PROGRAM PersonnelDoor
VAR
	
END_VAR

IF GVL_Doors.QQ1.OpenButtonRequestInput THEN
	GVL_Doors.QQ1.AccessAreaRequest := 1;
	GVL_Doors.QQ1.OpenButtonLED_Output := 1;
	GVL_Doors.QQ1.OkToUnlockDoor := 1; //Remove this once ventalation is hooked up. Ventalation and styrene sensor level will determine when this gets turned on.
	ELSE
	GVL_Doors.QQ1.OpenButtonLED_Output := 0;
END_IF

GVL_Doors.QQ1.OkToUnlockDoorRTRIG(CLK := GVL_Doors.QQ1.OkToUnlockDoor);


IF GVL_Doors.QQ1.OkToUnlockDoorRTRIG.Q THEN
	GVL_Doors.QQ1.AccessAreaRequest := 0;
	GVL_Doors.QQ1.OpenButtonLED_Output := 0;
	GVL_Doors.QQ1.LockButtonLED_Output := 1;
	GVL_Doors.QQ1.LockOutput := 1;
END_IF

IF GVL_Doors.QQ1.LockButtonRequestInput THEN
	GVL_Doors.QQ1.LockOutput := 0;	
	GVL_Doors.QQ1.LockButtonLED_Output := 0;
	GVL_Doors.QQ1.OkToUnlockDoor := 0; //Remove this once ventalation is hooked up.
END_IF

END_PROGRAM

(* stored: Version 1.1.0.1, ProductVersion 3.1.4024.12
   POU PersonnelDoor: Id {7b769278-a9dd-4399-a322-74769ac026ef}, SpecialFunc None *)
